{attribute 'GeneratedUsingTerminal: EL3312-0000-0018'}
{attribute addProperty BoxType "EL3312-0000-0018"}
{attribute addProperty Id "TC_Inputs_Channel_1AT %I*AI_Standard_Channel_4A3944819TC_Inputs_Channel_2AT %I*AI_Standard_Channel_4A3944819WcStateAT %I*WcState_9091E0EB2InfoDataAT %I*InfoData_32EB74EA10"}
{attribute addProperty CRC "3197676326"}
{attribute addProperty Size "30"}
TYPE EL3312_BE98AB26 EXTENDS EtcSlaveTerminalBase_947E5A46 :
STRUCT
	{attribute addProperty Name "TC_Inputs_Channel_1"}
	TC_Inputs_Channel_1 : AI_Standard_Channel_4A394481;
	{attribute addProperty Name "TC_Inputs_Channel_2"}
	TC_Inputs_Channel_2 : AI_Standard_Channel_4A394481;
	{attribute addProperty Name "WcState"}
	WcState : WcState_9091E0EB;
	{attribute addProperty Name "InfoData"}
	InfoData : InfoData_32EB74EA;
END_STRUCT
END_TYPE

(* stored: Version 1.2.0.0, ProductVersion 3.1.4024.9
   DUT EL3312_BE98AB26: Id {ebec33f6-ff1d-42da-a668-619a9c51a501} *)
